FUNCTION_BLOCK overcurrentV3_IO_1 (* Composite Function Block Type *)
  (* Standard: 61499-2 *)
  (* Version 0.0, 23/05/2016, Chen-Wei, nxtControl GmbH, template *)
  PACKAGE Main;
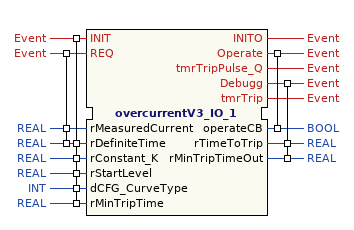
  EVENT_INPUT
    INIT WITH rDefiniteTime, rConstant_K, rStartLevel, dCFG_CurveType, rMinTripTime; (* Initialization Request *)
    REQ WITH rMeasuredCurrent, rDefiniteTime; (* Normal Execution Request *)
  END_EVENT
  EVENT_OUTPUT
    INITO; (* Initialization Confirm *)
    Operate WITH operateCB; (* Delayed Event *)
    tmrTripPulse_Q; (* Delayed Event *)
    Debugg WITH rTimeToTrip, rMinTripTimeOut;
    tmrTrip; (* Execution Confirmation *)
  END_EVENT
  VAR_INPUT
    rMeasuredCurrent : REAL; (* Input event qualifier *)
    rDefiniteTime : REAL;
    rConstant_K : REAL;
    rStartLevel : REAL;
    dCFG_CurveType : INT;
    rMinTripTime : REAL;
  END_VAR
  VAR_OUTPUT
    operateCB : BOOL; (* Output event qualifier *)
    rTimeToTrip : REAL;
    rMinTripTimeOut : REAL;
  END_VAR
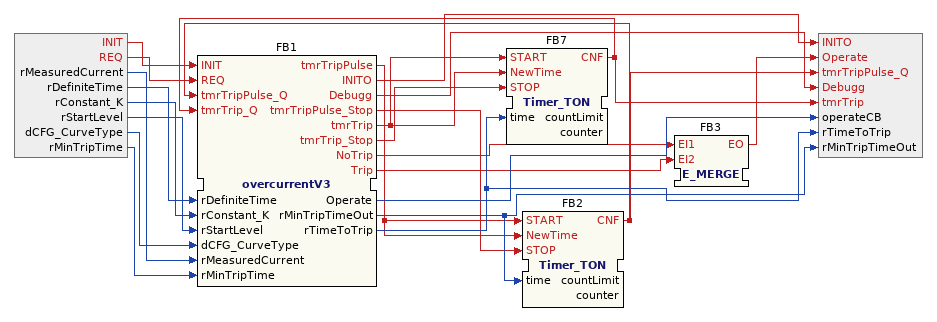
  FBS
    FB3 : E_MERGE;
    FB7 : Timer_TON;
    FB2 : Timer_TON;
    FB1 : overcurrentV3;
  END_FBS
  EVENT_CONNECTIONS
    INIT TO FB1.INIT;
    REQ TO FB1.REQ;
    FB1.tmrTripPulse TO FB2.START;
    FB2.CNF TO tmrTripPulse_Q;
    FB1.INITO TO INITO;
    FB1.Debugg TO Debugg;
    FB1.tmrTripPulse_Stop TO FB2.STOP;
    FB2.CNF TO FB1.tmrTripPulse_Q;
    FB1.tmrTrip TO FB7.NewTime;
    FB1.tmrTrip TO FB7.START;
    FB1.tmrTrip_Stop TO FB7.STOP;
    FB7.CNF TO FB1.tmrTrip_Q;
    FB7.CNF TO tmrTrip;
    FB1.tmrTripPulse TO FB2.NewTime;
    FB1.NoTrip TO FB3.EI1;
    FB1.Trip TO FB3.EI2;
    FB3.EO TO Operate;
  END_CONNECTIONS
  DATA_CONNECTIONS
    FB1.Operate TO operateCB;
    rDefiniteTime TO FB1.rDefiniteTime;
    rConstant_K TO FB1.rConstant_K;
    rStartLevel TO FB1.rStartLevel;
    dCFG_CurveType TO FB1.dCFG_CurveType;
    rMeasuredCurrent TO FB1.rMeasuredCurrent;
    FB1.rMinTripTimeOut TO FB2.time;
    FB1.rTimeToTrip TO rTimeToTrip;
    rMinTripTime TO FB1.rMinTripTime;
    FB1.rTimeToTrip TO FB7.time;
    FB1.rMinTripTimeOut TO rMinTripTimeOut;
  END_CONNECTIONS
END_FUNCTION_BLOCK
